INTERFACE I_State_Object

PROPERTY P_State : eObjectAktorState
GET
END_GET
END_PROPERTY

END_INTERFACE

(* stored: Version 1.1.0.1
   Itf I_State_Object: Id {e88975fe-9af3-41a3-bdeb-7dbbcbc10d6c}
   Property P_State: Id {ffc6be98-54b0-4146-b75d-41a68bad69c1}
   Get Get: Id {c2147764-6604-459b-af94-74bd8584b647} *)
